// TIA Portal V19 export
DATA_BLOCK "A0303_Manager_PERS"   // DB113
// stored: MemoryReserve 100
   VAR RETAIN
      Par : Struct
         Antiribaltamento : Struct
            Offset_Pos : LReal := 3.0;
         END_STRUCT;
      END_STRUCT;
   END_VAR
BEGIN
END_DATA_BLOCK
